# EPICS StreamDevice protocol: simulators/example/example.proto
# author: Ricardo Fernandes
# email: ricardo.fernandes@esss.se
# copyright: (C) 2015-2016 European Spallation Source (ESS)
# version: 1.0.2
# date: 2016/OCT/13
# description: File that describes the EPICS streamDevice protocol for the example simulator.

Terminator = CR LF;

get_power
{
   out "AC?";
   in "AC?%{0|1}";
}

set_power
{
   out "AC%{0|1}";
   @init {get_power};
}

get_fixed
{
   out "FIXED?";
   in "%f";
}

get_enum
{
   out "ENUM?";
   in "%d";
}

get_incr
{
   out "INCR?";
   in "%d";
}

get_random
{
   out "RANDOM?";
   in "%d";
}

get_custom
{
   out "CUSTOM1?";
   in "%f";
}
